Universal Robots PolyScope program: xmlrpc_example_posetrans.urp

Program xmlrpc_example_posetrans (installation=default directory=/programs/usbdisk createdIn=5.17.0 lastSavedIn=5.13.0 robotSerialNumber=20185300103)
Calibrated DH parameters: a=[-0.0001, -0.158233, -0.118758, 0.000117, -0.000141, 0]; d=[0.151763, 31.630685, -40.942779, 9.441239, 0.08534, 0.091753]; alpha=[1.570714, 0.005875, -0.018951, 1.571134, -1.571111, 0]; deltaTheta=[0, 0.865461, 6.396079, -0.978451, -0.000021, 0]
InitVariablesNode
BeforeStart
  'Configuración del XMLRPC'
  camera := rpc_factory("xmlrpc","http://192.168.23.147:50000")
  thetaY_camera_r := 1.13446
  reference_point := p[0,0.2,0.2,0,thetaY_camera_r,0]
Robot Program (runOnlyOnce=false)
  MoveJ speed 60 deg/s, acceleration 80 deg/s^2 (useActiveTCP=true) feature=Base
    Waypoint reference_p: TCP in base x=229.72 y=-205 z=17.553 mm, rx=0.8961 ry=-3.0111 rz=0 rad; joints [114.173, -53.943, 130.313, -166.371, -88.936, -9.818] deg; TCP offset x=0 y=0 z=30.6 mm, rx=0 ry=0 rz=0 rad
  next_pose := camera.get_next_pose()
  next_pose_list := p[next_pose[0],next_pose[1],next_pose[2],next_pose[3],next_pose[4],next_pose[5]]
  target := pose_trans(reference_p,next_pose_list)
  If next_pose[0] == 0 and next_pose[1] == 0
    MoveJ speed 60 deg/s, acceleration 80 deg/s^2 (useActiveTCP=true) feature=Base
      Waypoint Casa: TCP in base x=227.184 y=-42.646 z=302.891 mm, rx=-1.3425 ry=2.8169 rz=-0.0022 rad; joints [135.771, -114.961, 101.356, -76.885, -89.548, -6.253] deg
  Else 
    MoveP speed 50 mm/s, acceleration 80 mm/s^2 (blendRadius=0.025 useActiveTCP=true) feature=Base
      Waypoint Variable (Variable): variable=target
  Wait Sleep waitTime=1
